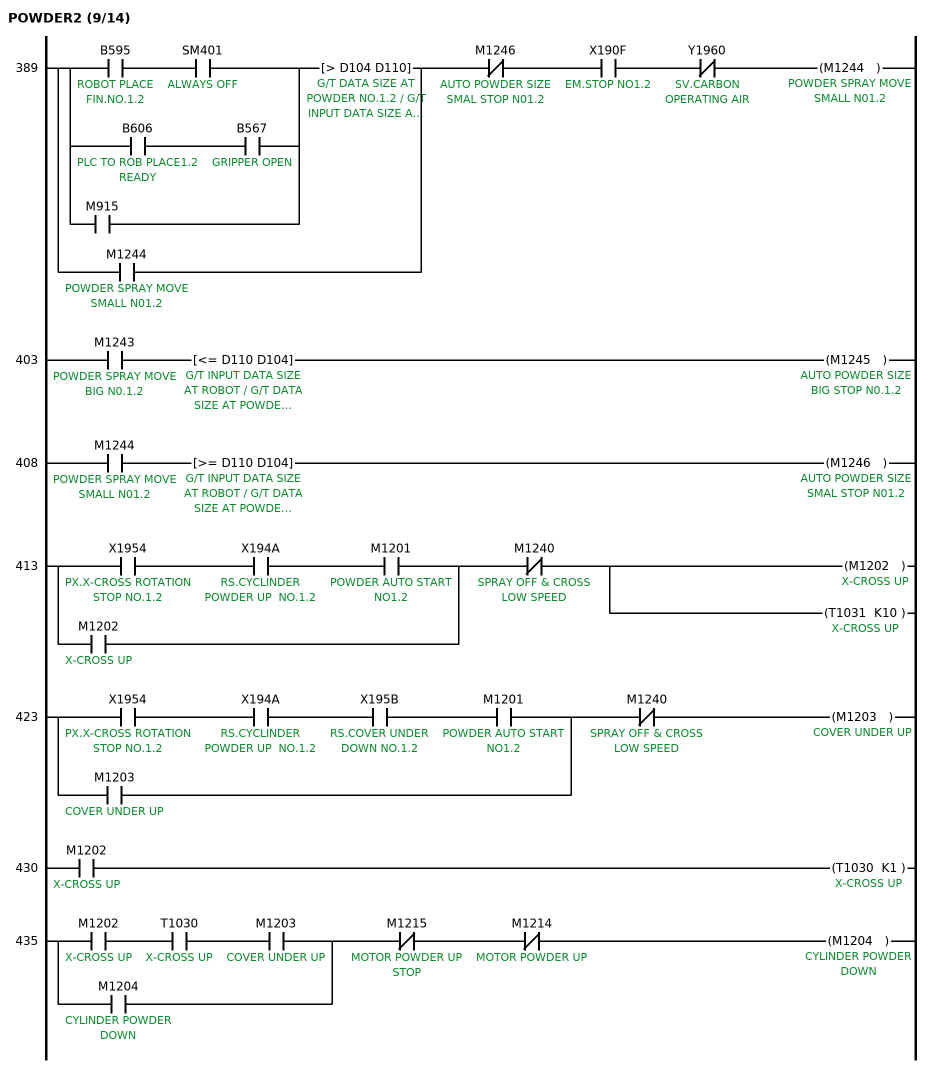
[picture p48: ladder of POWDER2, rungs at steps 389 to 435]
389   LD      B595  ; ROBOT PLACE FIN.NO.1.2
      AND     SM401  ; ALWAYS OFF
      LD      B606  ; PLC TO ROB PLACE1.2 READY
      AND     B567  ; GRIPPER OPEN
      ORB
      OR      M915
      AND>    D104 D110  ; G/T DATA SIZE AT POWDER NO.1.2 / G/T INPUT DATA SIZE AT ROBOT
      OR      M1244  ; POWDER SPRAY MOVE SMALL N01.2
      ANI     M1246  ; AUTO POWDER SIZE SMAL STOP N01.2
      AND     X190F  ; EM.STOP NO1.2
      ANI     Y1960  ; SV.CARBON OPERATING AIR
      OUT     M1244  ; POWDER SPRAY MOVE SMALL N01.2
403   LD      M1243  ; POWDER SPRAY MOVE  BIG N0.1.2
      AND<=   D110 D104  ; G/T INPUT DATA SIZE AT ROBOT / G/T DATA SIZE AT POWDER NO.1.2
      OUT     M1245  ; AUTO POWDER SIZE BIG STOP N0.1.2
408   LD      M1244  ; POWDER SPRAY MOVE SMALL N01.2
      AND>=   D110 D104  ; G/T INPUT DATA SIZE AT ROBOT / G/T DATA SIZE AT POWDER NO.1.2
      OUT     M1246  ; AUTO POWDER SIZE SMAL STOP N01.2
413   LD      X1954  ; PX.X-CROSS ROTATION STOP NO.1.2
      AND     X194A  ; RS.CYCLINDER POWDER UP  NO.1.2
      AND     M1201  ; POWDER AUTO START NO1.2
      OR      M1202  ; X-CROSS UP
      ANI     M1240  ; SPRAY OFF & CROSS LOW SPEED
      OUT     M1202  ; X-CROSS UP
      OUT     T1031 K10  ; X-CROSS UP
423   LD      X1954  ; PX.X-CROSS ROTATION STOP NO.1.2
      AND     X194A  ; RS.CYCLINDER POWDER UP  NO.1.2
      AND     X195B  ; RS.COVER UNDER DOWN NO.1.2
      AND     M1201  ; POWDER AUTO START NO1.2
      OR      M1203  ; COVER UNDER UP
      ANI     M1240  ; SPRAY OFF & CROSS LOW SPEED
      OUT     M1203  ; COVER UNDER UP
430   LD      M1202  ; X-CROSS UP
      OUT     T1030 K1  ; X-CROSS UP
435   LD      M1202  ; X-CROSS UP
      AND     T1030  ; X-CROSS UP
      AND     M1203  ; COVER UNDER UP
      OR      M1204  ; CYLINDER POWDER DOWN
      ANI     M1215  ; MOTOR POWDER UP STOP
      ANI     M1214  ; MOTOR POWDER UP
      OUT     M1204  ; CYLINDER POWDER DOWN
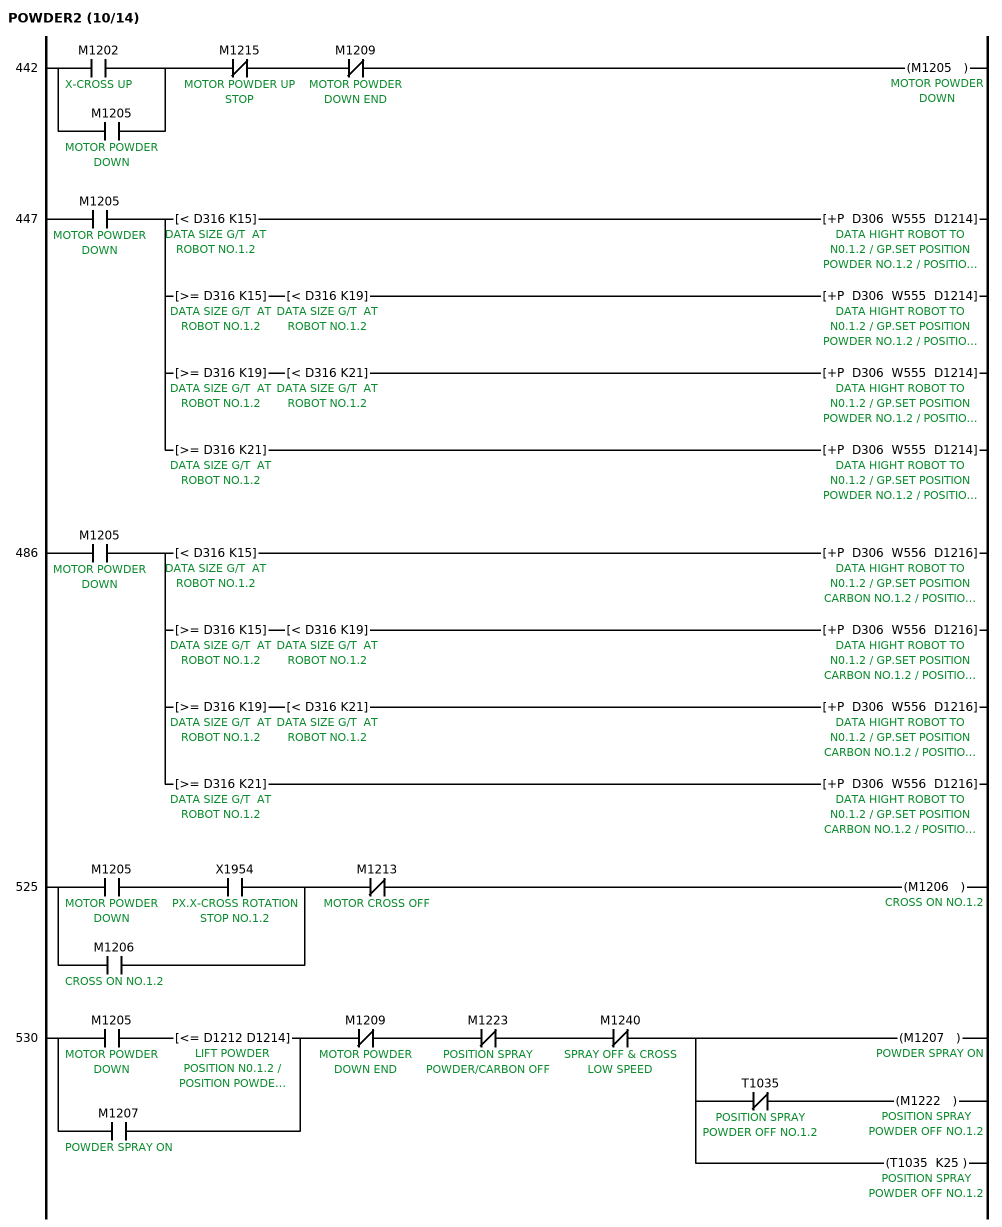
442   LD      M1202  ; X-CROSS UP
      OR      M1205  ; MOTOR POWDER DOWN
      ANI     M1215  ; MOTOR POWDER UP STOP
      ANI     M1209  ; MOTOR POWDER DOWN END
      OUT     M1205  ; MOTOR POWDER DOWN
447   LD      M1205  ; MOTOR POWDER DOWN
      MPS
      AND<    D316 K15  ; DATA SIZE G/T  AT ROBOT NO.1.2
      +P      D306 W555 D1214  ; GP.SET POSITION POWDER NO.1.2 / POSITION POWDER SPRAY ON NO.1.2
      MRD
      AND>=   D316 K15  ; DATA SIZE G/T  AT ROBOT NO.1.2
      AND<    D316 K19  ; DATA SIZE G/T  AT ROBOT NO.1.2
      +P      D306 W555 D1214
      MRD
      AND>=   D316 K19  ; DATA SIZE G/T  AT ROBOT NO.1.2
      AND<    D316 K21  ; DATA SIZE G/T  AT ROBOT NO.1.2
      +P      D306 W555 D1214
      MPP
      AND>=   D316 K21  ; DATA SIZE G/T  AT ROBOT NO.1.2
      +P      D306 W555 D1214
486   LD      M1205  ; MOTOR POWDER DOWN
      MPS
      AND<    D316 K15  ; DATA SIZE G/T  AT ROBOT NO.1.2
      +P      D306 W556 D1216  ; GP.SET POSITION CARBON NO.1.2 / POSITION CARBON ON NO.1.2
      MRD
      AND>=   D316 K15  ; DATA SIZE G/T  AT ROBOT NO.1.2
      AND<    D316 K19  ; DATA SIZE G/T  AT ROBOT NO.1.2
      +P      D306 W556 D1216
      MRD
      AND>=   D316 K19  ; DATA SIZE G/T  AT ROBOT NO.1.2
      AND<    D316 K21  ; DATA SIZE G/T  AT ROBOT NO.1.2
      +P      D306 W556 D1216
      MPP
      AND>=   D316 K21  ; DATA SIZE G/T  AT ROBOT NO.1.2
      +P      D306 W556 D1216
525   LD      M1205  ; MOTOR POWDER DOWN
      AND     X1954  ; PX.X-CROSS ROTATION STOP NO.1.2
      OR      M1206  ; CROSS ON NO.1.2
      ANI     M1213  ; MOTOR CROSS OFF
      OUT     M1206  ; CROSS ON NO.1.2
530   LD      M1205  ; MOTOR POWDER DOWN
      AND<=   D1212 D1214  ; LIFT POWDER POSITION N0.1.2 / POSITION POWDER SPRAY ON NO.1.2
      OR      M1207  ; POWDER SPRAY ON
      ANI     M1209  ; MOTOR POWDER DOWN END
      ANI     M1223  ; POSITION SPRAY POWDER/CARBON OFF
      ANI     M1240  ; SPRAY OFF & CROSS LOW SPEED
      OUT     M1207  ; POWDER SPRAY ON
      MPS
      ANI     T1035  ; POSITION SPRAY POWDER OFF NO.1.2
      OUT     M1222  ; POSITION SPRAY POWDER OFF NO.1.2
      MPP
      OUT     T1035 K25  ; POSITION SPRAY POWDER OFF NO.1.2
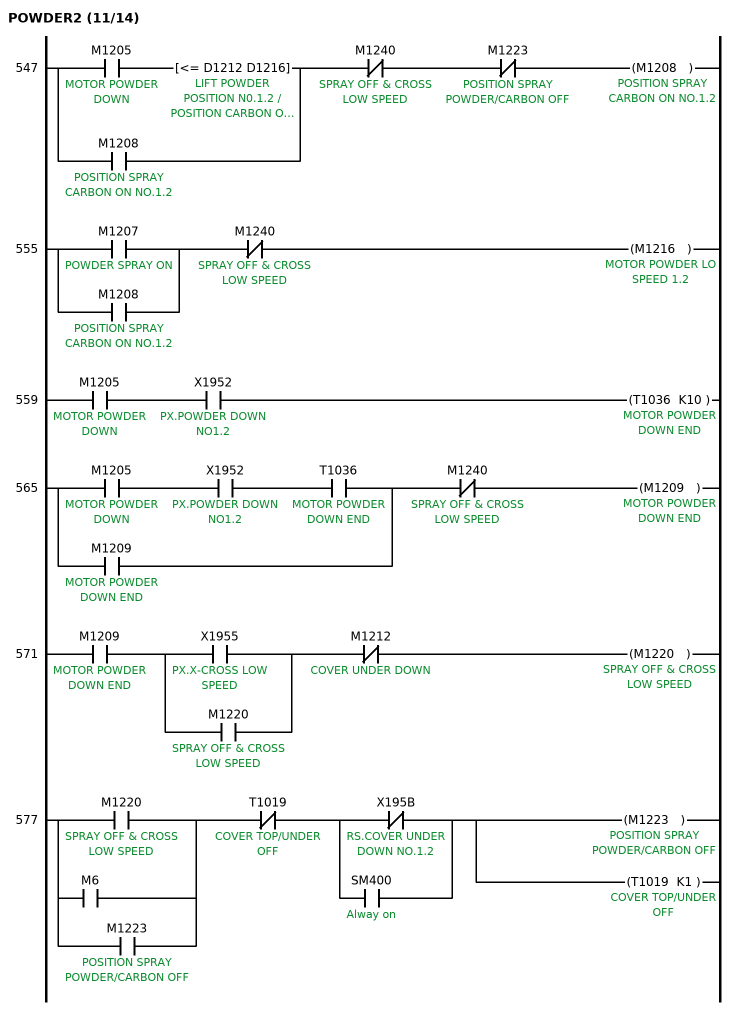
547   LD      M1205  ; MOTOR POWDER DOWN
      AND<=   D1212 D1216  ; LIFT POWDER POSITION N0.1.2 / POSITION CARBON ON NO.1.2
      OR      M1208  ; POSITION SPRAY CARBON ON NO.1.2
      ANI     M1240  ; SPRAY OFF & CROSS LOW SPEED
      ANI     M1223  ; POSITION SPRAY POWDER/CARBON OFF
      OUT     M1208  ; POSITION SPRAY CARBON ON NO.1.2
555   LD      M1207  ; POWDER SPRAY ON
      OR      M1208  ; POSITION SPRAY CARBON ON NO.1.2
      ANI     M1240  ; SPRAY OFF & CROSS LOW SPEED
      OUT     M1216  ; MOTOR POWDER LO SPEED 1.2
559   LD      M1205  ; MOTOR POWDER DOWN
      AND     X1952  ; PX.POWDER DOWN NO1.2
      OUT     T1036 K10  ; MOTOR POWDER DOWN END
565   LD      M1205  ; MOTOR POWDER DOWN
      AND     X1952  ; PX.POWDER DOWN NO1.2
      AND     T1036  ; MOTOR POWDER DOWN END
      OR      M1209  ; MOTOR POWDER DOWN END
      ANI     M1240  ; SPRAY OFF & CROSS LOW SPEED
      OUT     M1209  ; MOTOR POWDER DOWN END
571   LD      M1209  ; MOTOR POWDER DOWN END
      LD      X1955  ; PX.X-CROSS LOW SPEED
      OR      M1220  ; SPRAY OFF & CROSS LOW SPEED
      ANB
      ANI     M1212  ; COVER UNDER DOWN
      OUT     M1220  ; SPRAY OFF & CROSS LOW SPEED
577   LD      M1220  ; SPRAY OFF & CROSS LOW SPEED
      OR      M6
      OR      M1223  ; POSITION SPRAY POWDER/CARBON OFF
      ANI     T1019  ; COVER TOP/UNDER OFF
      LDI     X195B  ; RS.COVER UNDER DOWN NO.1.2
      OR      SM400  ; Alway on
      ANB
      OUT     M1223  ; POSITION SPRAY POWDER/CARBON OFF
      OUT     T1019 K1  ; COVER TOP/UNDER OFF
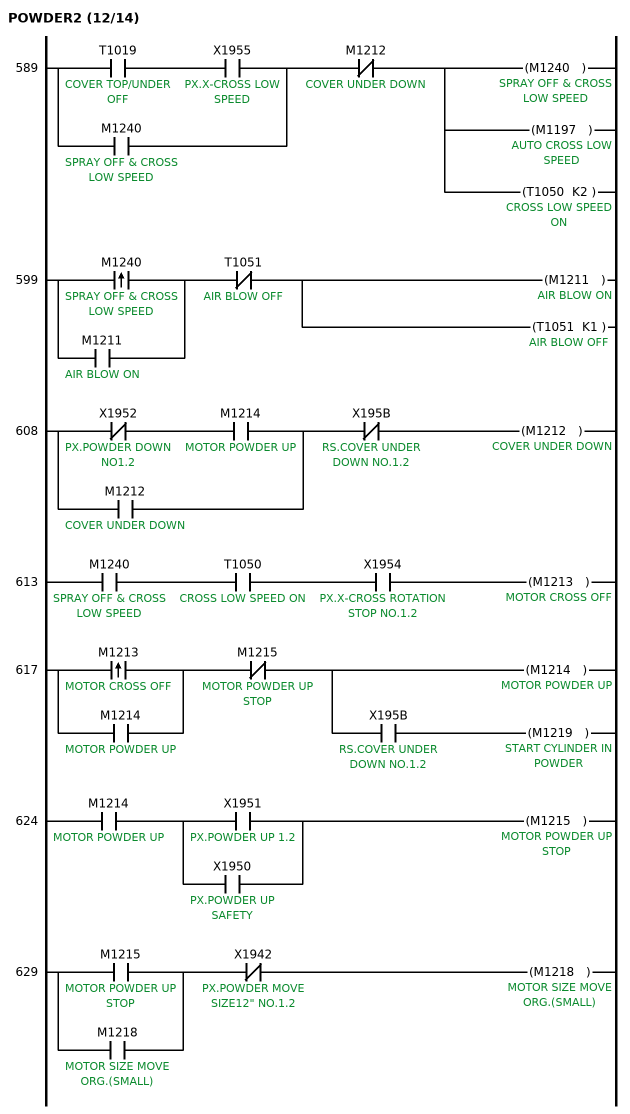
589   LD      T1019  ; COVER TOP/UNDER OFF
      AND     X1955  ; PX.X-CROSS LOW SPEED
      OR      M1240  ; SPRAY OFF & CROSS LOW SPEED
      ANI     M1212  ; COVER UNDER DOWN
      OUT     M1240  ; SPRAY OFF & CROSS LOW SPEED
      OUT     M1197  ; AUTO CROSS LOW SPEED
      OUT     T1050 K2  ; CROSS LOW SPEED ON
599   LDP     M1240  ; SPRAY OFF & CROSS LOW SPEED
      OR      M1211  ; AIR BLOW ON
      ANI     T1051  ; AIR BLOW OFF
      OUT     M1211  ; AIR BLOW ON
      OUT     T1051 K1  ; AIR BLOW OFF
608   LDI     X1952  ; PX.POWDER DOWN NO1.2
      AND     M1214  ; MOTOR POWDER UP
      OR      M1212  ; COVER UNDER DOWN
      ANI     X195B  ; RS.COVER UNDER DOWN NO.1.2
      OUT     M1212  ; COVER UNDER DOWN
613   LD      M1240  ; SPRAY OFF & CROSS LOW SPEED
      AND     T1050  ; CROSS LOW SPEED ON
      AND     X1954  ; PX.X-CROSS ROTATION STOP NO.1.2
      OUT     M1213  ; MOTOR CROSS OFF
617   LDP     M1213  ; MOTOR CROSS OFF
      OR      M1214  ; MOTOR POWDER UP
      ANI     M1215  ; MOTOR POWDER UP STOP
      OUT     M1214  ; MOTOR POWDER UP
      AND     X195B  ; RS.COVER UNDER DOWN NO.1.2
      OUT     M1219  ; START CYLINDER IN POWDER
624   LD      M1214  ; MOTOR POWDER UP
      LD      X1951  ; PX.POWDER UP 1.2
      OR      X1950  ; PX.POWDER UP SAFETY
      ANB
      OUT     M1215  ; MOTOR POWDER UP STOP
629   LD      M1215  ; MOTOR POWDER UP STOP
      OR      M1218  ; MOTOR SIZE MOVE ORG.(SMALL)
      ANI     X1942  ; PX.POWDER MOVE SIZE12" NO.1.2
      OUT     M1218  ; MOTOR SIZE MOVE ORG.(SMALL)
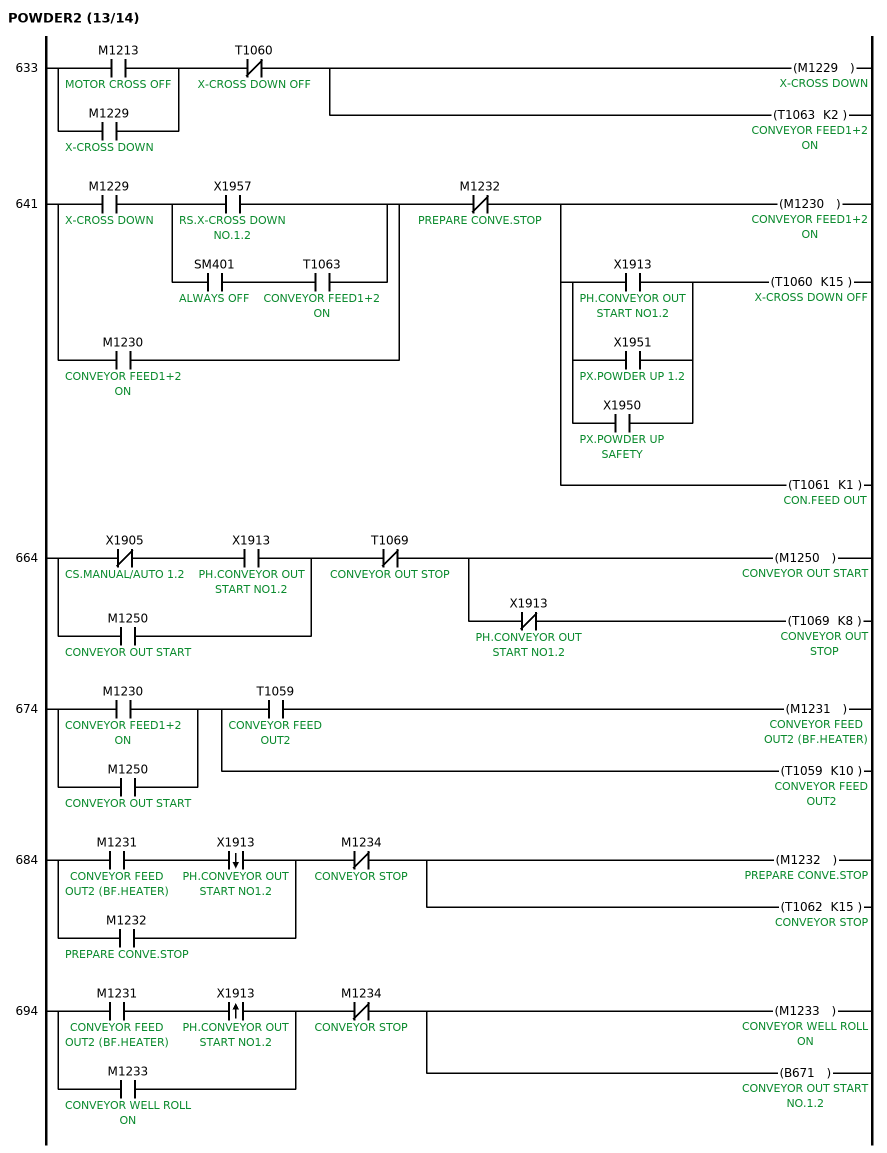
633   LD      M1213  ; MOTOR CROSS OFF
      OR      M1229  ; X-CROSS DOWN
      ANI     T1060  ; X-CROSS DOWN OFF
      OUT     M1229  ; X-CROSS DOWN
      OUT     T1063 K2  ; CONVEYOR FEED1+2 ON
641   LD      M1229  ; X-CROSS DOWN
      LD      X1957  ; RS.X-CROSS DOWN NO.1.2
      LD      SM401  ; ALWAYS OFF
      AND     T1063  ; CONVEYOR FEED1+2 ON
      ORB
      ANB
      OR      M1230  ; CONVEYOR FEED1+2 ON
      ANI     M1232  ; PREPARE CONVE.STOP
      OUT     M1230  ; CONVEYOR FEED1+2 ON
      MPS
      LD      X1913  ; PH.CONVEYOR OUT START NO1.2
      OR      X1951  ; PX.POWDER UP 1.2
      OR      X1950  ; PX.POWDER UP SAFETY
      ANB
      OUT     T1060 K15  ; X-CROSS DOWN OFF
      MPP
      OUT     T1061 K1  ; CON.FEED OUT
664   LDI     X1905  ; CS.MANUAL/AUTO 1.2
      AND     X1913  ; PH.CONVEYOR OUT START NO1.2
      OR      M1250  ; CONVEYOR OUT START
      ANI     T1069  ; CONVEYOR OUT STOP
      OUT     M1250  ; CONVEYOR OUT START
      ANI     X1913  ; PH.CONVEYOR OUT START NO1.2
      OUT     T1069 K8  ; CONVEYOR OUT STOP
674   LD      M1230  ; CONVEYOR FEED1+2 ON
      OR      M1250  ; CONVEYOR OUT START
      MPS
      AND     T1059  ; CONVEYOR FEED OUT2
      OUT     M1231  ; CONVEYOR FEED OUT2 (BF.HEATER)
      MPP
      OUT     T1059 K10  ; CONVEYOR FEED OUT2
684   LD      M1231  ; CONVEYOR FEED OUT2 (BF.HEATER)
      ANDF    X1913  ; PH.CONVEYOR OUT START NO1.2
      OR      M1232  ; PREPARE CONVE.STOP
      ANI     M1234  ; CONVEYOR STOP
      OUT     M1232  ; PREPARE CONVE.STOP
      OUT     T1062 K15  ; CONVEYOR STOP
694   LD      M1231  ; CONVEYOR FEED OUT2 (BF.HEATER)
      ANDP    X1913  ; PH.CONVEYOR OUT START NO1.2
      OR      M1233  ; CONVEYOR WELL ROLL ON
      ANI     M1234  ; CONVEYOR STOP
      OUT     M1233  ; CONVEYOR WELL ROLL ON
      OUT     B671  ; CONVEYOR OUT START NO.1.2
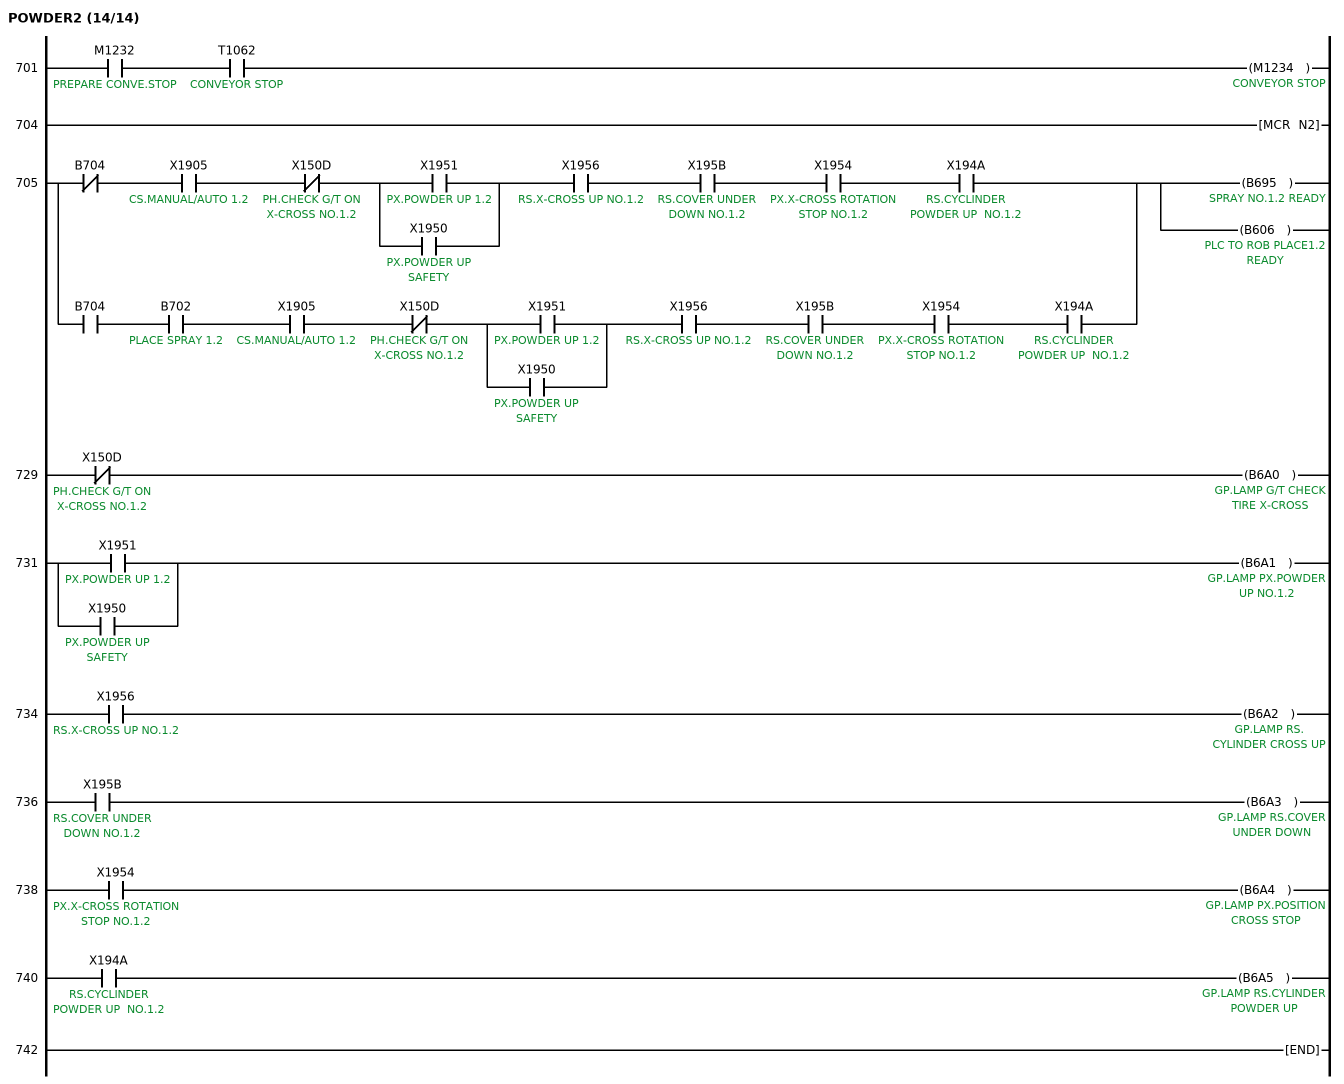
701   LD      M1232  ; PREPARE CONVE.STOP
      AND     T1062  ; CONVEYOR STOP
      OUT     M1234  ; CONVEYOR STOP
704   MCR     N2
705   LDI     B704
      AND     X1905  ; CS.MANUAL/AUTO 1.2
      ANI     X150D  ; PH.CHECK G/T ON X-CROSS NO.1.2
      LD      X1951  ; PX.POWDER UP 1.2
      OR      X1950  ; PX.POWDER UP SAFETY
      ANB
      AND     X1956  ; RS.X-CROSS UP NO.1.2
      AND     X195B  ; RS.COVER UNDER DOWN NO.1.2
      AND     X1954  ; PX.X-CROSS ROTATION STOP NO.1.2
      AND     X194A  ; RS.CYCLINDER POWDER UP  NO.1.2
      LD      B704
      AND     B702  ; PLACE SPRAY 1.2
      AND     X1905  ; CS.MANUAL/AUTO 1.2
      ANI     X150D  ; PH.CHECK G/T ON X-CROSS NO.1.2
      LD      X1951  ; PX.POWDER UP 1.2
      OR      X1950  ; PX.POWDER UP SAFETY
      ANB
      AND     X1956  ; RS.X-CROSS UP NO.1.2
      AND     X195B  ; RS.COVER UNDER DOWN NO.1.2
      AND     X1954  ; PX.X-CROSS ROTATION STOP NO.1.2
      AND     X194A  ; RS.CYCLINDER POWDER UP  NO.1.2
      ORB
      OUT     B695  ; SPRAY NO.1.2 READY
      OUT     B606  ; PLC TO ROB PLACE1.2 READY
729   LDI     X150D  ; PH.CHECK G/T ON X-CROSS NO.1.2
      OUT     B6A0  ; GP.LAMP G/T CHECK TIRE X-CROSS
731   LD      X1951  ; PX.POWDER UP 1.2
      OR      X1950  ; PX.POWDER UP SAFETY
      OUT     B6A1  ; GP.LAMP PX.POWDER UP NO.1.2
734   LD      X1956  ; RS.X-CROSS UP NO.1.2
      OUT     B6A2  ; GP.LAMP RS. CYLINDER CROSS UP
736   LD      X195B  ; RS.COVER UNDER DOWN NO.1.2
      OUT     B6A3  ; GP.LAMP RS.COVER UNDER DOWN
738   LD      X1954  ; PX.X-CROSS ROTATION STOP NO.1.2
      OUT     B6A4  ; GP.LAMP PX.POSITION CROSS STOP
740   LD      X194A  ; RS.CYCLINDER POWDER UP  NO.1.2
      OUT     B6A5  ; GP.LAMP RS.CYLINDER POWDER UP
742   END
END_PROGRAM

PROGRAM 62DA
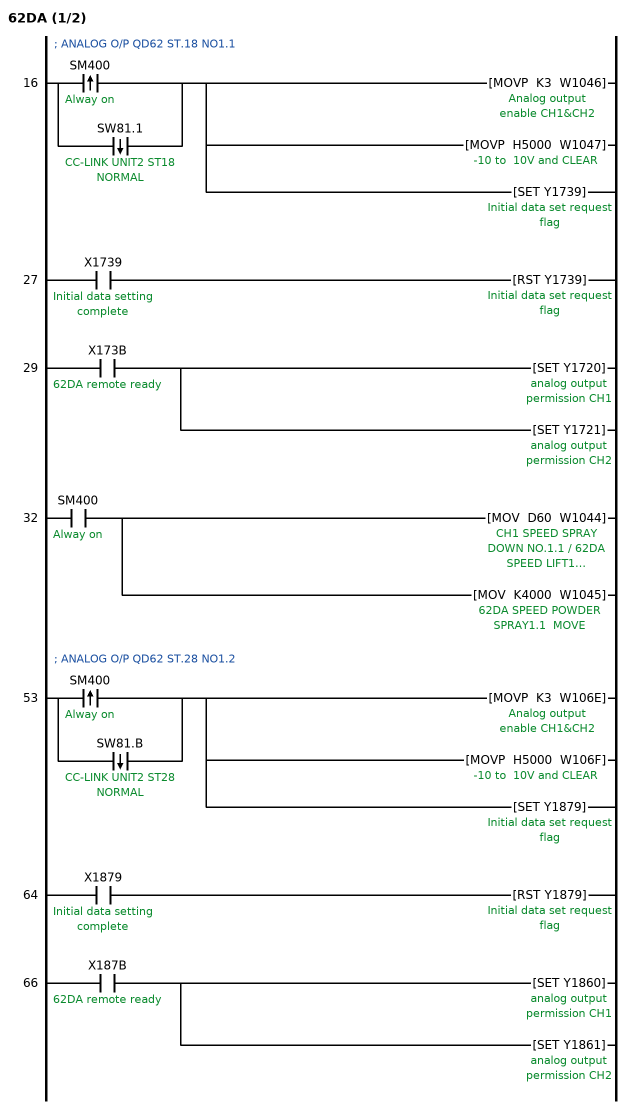
; ANALOG O/P QD62 ST.18 NO1.1
16    LDP     SM400  ; Alway on
      ORF     SW81.1  ; CC-LINK UNIT2 ST18 NORMAL
      MOVP    K3 W1046  ; Analog output enable CH1&CH2
      MOVP    H5000 W1047  ; -10 to  10V and CLEAR
      SET     Y1739  ; Initial data set request flag
27    LD      X1739  ; Initial data setting complete
      RST     Y1739  ; Initial data set request flag
29    LD      X173B  ; 62DA remote ready
      SET     Y1720  ; analog output permission CH1
      SET     Y1721  ; analog output permission CH2
32    LD      SM400  ; Alway on
      MOV     D60 W1044  ; CH1 SPEED SPRAY DOWN NO.1.1 / 62DA SPEED LIFT1.1POWDER UP/DOWN
      MOV     K4000 W1045  ; 62DA SPEED POWDER SPRAY1.1  MOVE
; ANALOG O/P QD62 ST.28 NO1.2
53    LDP     SM400  ; Alway on
      ORF     SW81.B  ; CC-LINK UNIT2 ST28 NORMAL
      MOVP    K3 W106E  ; Analog output enable CH1&CH2
      MOVP    H5000 W106F  ; -10 to  10V and CLEAR
      SET     Y1879  ; Initial data set request flag
64    LD      X1879  ; Initial data setting complete
      RST     Y1879  ; Initial data set request flag
66    LD      X187B  ; 62DA remote ready
      SET     Y1860  ; analog output permission CH1
      SET     Y1861  ; analog output permission CH2
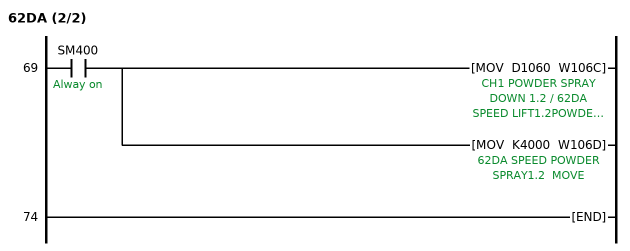
69    LD      SM400  ; Alway on
      MOV     D1060 W106C  ; CH1 POWDER SPRAY DOWN 1.2 / 62DA SPEED LIFT1.2POWDER UP/DOWN
      MOV     K4000 W106D  ; 62DA SPEED POWDER SPRAY1.2  MOVE
74    END
END_PROGRAM

// 3 SFC block(s) not rendered

// device comments not shown above
X109  ; GRIPPER BWD 2
X10B  ; GRIPPER BWD 4
X10C  ; GRIPPER BWD 5
X10D  ; GRIPPER BWD 6
X10A0  ; SIZE 21
X10A1  ; SENSOR 2
X10A2  ; SENSOR 3
X10A3  ; SIZE 12
X152A  ; ROBOT HOEM END
X152B  ; OFF CARBON
X152F  ; CC-LINK BIT RECEIVE ROBOT
X1530  ; ROBOT DATA REQUEST
X1531  ; ROBOT DATA RECIEVED
X1532  ; ROBOT STADBLY
X1533  ; ROBOT PICK POINT RDY.
X1534  ; ROBOT UO FIN.
X1537  ; ROBOT PLACE FIN
X1538  ; ROBOT SAFTY POINT
X153A  ; ROBOT SPARY COMPLETED
X153D  ; SPRAY NO.6  START
X153E  ; SPRAY NO.5  START
X16C3  ; PH. SENSOR( IN2 CV)
X16E6  ; PH. SENSOR( IN1 CV) FULL
X16E7  ; PH. SENSOR(END CV)
X16E8  ; SS.CHECK TIRE ON X-CROSS
X16EA  ; RS.GRIPPER ORG.
X1738  ; Initial data processing request
X17D0  ; PH.CONV.AFTER HEATER
X1800  ; EMG.STOP
X180B  ; RS.CYCLINDER POWDER DOWN
X1818  ; RS.COVER TOP UP
X1819  ; RS.COVER TOP DOWN
X181A  ; RS.COVER UNDER UP
X1878  ; Initial data processing request
X194B  ; RS.CYCLINDER POWDER DOWN
X1958  ; RS.COVER TOP UP
X1959  ; RS.COVER TOP DOWN
X195A  ; RS.COVER UNDER UP
Y124  ; INVERTER MAGNETIC
Y125  ; inverter run
Y150  ; SERVO RUN
Y1020  ; INV.CONVEYOR IN FOR.
Y1021  ; INV.CONVEYOR IN REV.
Y1022  ; INV.CONVEYOR IN HI.
Y1023  ; INV.CONVEYOR IN LOW.
Y1024  ; INV.CONVEYOR OUT1 FOR.
Y1025  ; INV.CONVEYOR OUT REV.
Y1026  ; INV.CONVEYOR OUT HI.
Y1027  ; INV.CONVEYOR OUT LOW.
Y1028  ; INV.X-CROSS FOR.
Y1029  ; INV.X-CROSS REV.
Y102A  ; INV.X-CROSS HI.
Y102B  ; INV.X-CROSS LOW.
Y102C  ; MG.CONVEYOR REAR
Y102D  ; MG.BLOWER
Y102E  ; RY.MOTOR X-CROSS BREAK
Y102F  ; SV.POWDER SPRAY ON
Y1030  ; SV.CARBON SPRAY ON
Y1031  ; SV.CARBON SPRAY ATOMIZING HI
Y1032  ; SV.CARBON SPRAY ATOMIZING LOW
Y1033  ; SV.POWDER SPRAY ATOMIZING
Y1034  ; SV.X-CROSS UP/DOWN
Y1035  ; SV.BRAKE X-CROSS
Y1037  ; INV.CONVEYOR AFTER HEATER
Y1039  ; RY.CONV. HEATER
Y103A  ; RY.FAN CONVEYOR BEFORE HEATER
Y103B  ; RY.TEMP.HEATER ON
Y103C  ; MG.BLOWER HEATER
Y1511  ; MG.FILTER POWDER
Y1515  ; ROTATION
Y1516  ; VACCUM
Y151D  ; FWD
Y151E  ; BWD
Y152A  ; ROBOT HOME
Y1531  ; DATA XYZ WRITE
Y1534  ; GRIPPER FIN
Y1535  ; SPRAY NO.1.1 REQ.
Y1536  ; SPRAY NO.1.2 REQ.
Y1537  ; WORK REQUEST
Y1538  ; ROBOT SAFTY POINT( START SPAY)
Y1539  ; GRIPPER SAFTY ZONE COMPLETED
Y153A  ; ROBOT Z-AXIS START
Y153B  ; SPRAY COMPLETED STOP
Y16AD  ; SOL.LIFTER DOWN
Y16AE  ; HI-ROTOR ROTATE
Y16AF  ; HI-ROTOR ORG
Y1878  ; Initial data process complete
M12  ; PROTECT LIFT UP
M20  ; SW.MAN/AUTO
M150  ; CONVEYOR OUT START
M500  ; SW.AUTO
M501  ; POWDER AUTO START
M503  ; PREPARE SPRAY ON
M505  ; SPRAY CARBON ON
M506  ; SPRAY END
M507  ; ROTATION LOW SPEED
M508  ; ROTATION STOP
M510  ; CONVEYOR FEED1+2 ON
M511  ; CONVEYOR FEED OUT2
M512  ; PREPARE CONVE.STOP
M513  ; CONVEYOR WELL ROLL ON
M520  ; CONV. NO.4 WELL ROLL
M530  ; MANUAL X-CROSS ON
M531  ; MANUAL X-CROSS LOW
M532  ; MANUAL X-CROSS STOP
M550  ; STEP AUTO
M601  ; GP.CONVEYOR FEED OUT1
M602  ; GP.CONVEYOR FEED OUT2
M604  ; GP.X-CROSS UP
M606  ; CONVEYOR WELL ROLL NO1.
M607  ; CONVEYOR WELL ROLL NO2.
M608  ; CONVEYOR WELL ROLL NO3.
M609  ; CONVEYOR WELL ROLL NO4.
M801  ; LED-L ERROR
M805  ; SHUTTER EMG
M806  ; SHUTTER EMG
M910  ; NO USE
M955  ; TEST FAN CONVEYOR HEATER
M1000  ; AUTO MODE
M1003  ; GRIPPER HOME START
M1007  ; GRIPPER HOME END
M1008  ; CHECK SIZE 21"
M1053  ; GP.POWDER AUTO START
M1103  ; START OPEN(2)
M1110  ; WRITE DATA TO ROBOT
M1111  ; DATA GRIPPER
M1112  ; GRIPPER CLOSE START
M1114  ; GRIPPER CLOSE
M1118  ; START OPEN
M1119  ; Z-SPEED WRITE
M1200  ; SPRAY
M1300  ; lifter unit
B102  ; ERROR RESET(GOT)
B103  ; GP.CAMERA TRIGGER
B104  ; R-OFF RUBBER
B111  ; 13"
B112  ; 14"
B113  ; 15"
B114  ; 16"
B115  ; 17"
B116  ; 18"
B117  ; 19"
B118  ; 21"
B121  ; WRITE
B203  ; START(GOT)
B204  ; SERVO STOP
B205  ; GP.SERVO GRIPPER HOME
B208  ; SERVO VACCUM
B210  ; GP.SERVO GRIPPER JOG CLOSE
B211  ; GP.SERVO GRIPPER JOG OPEN
B312  ; GP.HEATER ON
B313  ; GP.HEATER OFF
B314  ; GP.BLOWER HEATER ON
B315  ; GP.BLOWER HEATER OFF
B321  ; GP.CONVEYOR FEED IN STOP
B323  ; GP.CONVEYOR FEED OUT1 STOP
B326  ; GP.CONVEYOR FEED OUT2 STOP
B328  ; GP.CONVEYOR HEATER STOP
B32A  ; GP.CONVEYOR NO3,4 WELLROLL STOP
B32B  ; GP.POWDER SPRAY ON
B32C  ; GP.CARBON SPRAY ON
B32E  ; GP.DUST COLLECTOR ON
B32F  ; GP.DUST COLLECTOR OFF
B692  ; DATA RECIEVED NO.6
B6C0  ; CHECK SIZE GRIPPER
B1000  ; JOG-
B1001  ; JOG+
B1002  ; SERVO ON
B1003  ; SERVO OFF
B1007  ; EROR RESET
B1010  ; JOG-
B1011  ; JOG+
B1012  ; SERVO ON
B1013  ; SERVO OFF
B1017  ; ERROR RESET
B1020  ; TEACH 1
B1023  ; TEACH
B1024  ; TEACH
B1030  ; TEACH 1
B1032  ; TEACH 3
T1  ; CONVE.FEED OUT
T3  ; CONVEYOR FEED1+2 ON
T4  ; CONV. NO.4 WELL ROLL OFF
T5  ; SPRAY END
T10  ; RESET AUTO STEP
T15  ; SW.MANUAL ON
T19  ; CONVEYOR FEED OUT2
T40  ; TIME SAFTY CYLINDER FWD
T120  ; DATA WRITE DELAY
T121  ; DATA TRANSFER DELAY
T150  ; CROSS LOW SPEED ON
T222  ; GRIPPER CLOSE DELAY
T250  ; GP.SPRAY POWDER ON
T251  ; GP.SPRAY CARBON ON
T252  ; ROBOT DOWN
T299  ; NO USE
T300  ; TRIGGER DELAY
T320  ; GRIPPER DELAY
T321  ; GRIPPER DELAY 21"
T420  ; DATA WRITE
T422  ; WRITE DATA DELAY
T430  ; rubber sensor
T444  ; PROTECT LIFT UP
T615  ; VACCUM OFF TIME
T720  ; 17-19 inch
T721  ; 21 inch
T722  ; 14 inch
D210  ; GP.POSITION SPRAY ON
D240  ; TRANSFER DATA
D300  ; RUBBER HIGHT ( DATA MEMOMY)
D310  ; RUBBER DIAMETER(DATA MEMORY)
D540  ; = D200 K0
D900  ; 64AD UNIT6 ERROR CODE
D1500  ; GP.SPRAY ADJUST POSITION
D2000  ; GRIPPER CLOSE DATA
D2002  ; OPEN DTA
D2100  ; SAFTY ZONE GRIPPER
D2200  ; OPEN POINT BEFORE PICK
D3100  ; POS.1
D3102  ; POS.2
D3104  ; POS.3
D3106  ; POS.4
D3108  ; EJECT POINT
D3212  ; SPRAY CARBON ON
D3300  ; BWD POSITION
D3302  ; EJECT POINT
D3304  ; POS.3
D3990  ; GRIPPER DELAY
D6000  ; DATA CAMERA DIAMERTER
D6002  ; Y-POSITION
D6004  ; X-POSITION
D6006  ; Z-POSITION
D7000  ; Position address/movement No1.
D7002  ; Command speed No1.
D7004  ; Position address/movement No2.
D7006  ; Command speed No2.
D7020  ; POSITION ADDDRESS
D7050  ; Axis 1 JOG SPEED
D7400  ; GP.Current feed value
D7500  ; GP.ROBOT SPRAY SPEED
W690  ; DATA HEIGHT TO POWDER NO.6
W695  ; DATA HEIGHT TO POWDER NO.5
W1000  ; POSITION ROBOT
W1006  ; Y-POSITION
W100E  ; DATA TO ROBOT SPRAY SPEED
W1014  ; TARGETPOSITION
W1016  ; POSITION WIDTH
W101E  ; ACC
W101F  ; DEC
W1021  ; LOAD CURRENT
W1024  ; TARGET POSITION
W1026  ; POSITION WIDTH
W102E  ; ACC
W102F  ; DEC
W1031  ; LOAD CURRENT
W1514  ; CURRENT POSITION
W1524  ; CURRENT POSITION
W1544  ; CH1 POWDER SPRAY DOWN
W156C  ; CH1 POWDER SPRAY DOWN
BL3  ; LIFTER
W200.8  ; CC_LINK ST1 ENABLE
W214.8  ; CC_LINK ST2 ENABLE
W228.8  ; CC_LINK ST3 ENABLE
W23C.8  ; CC_LINK ST4 ENABLE
